Universal Robots PolyScope program: cb_pulley_v3.urp

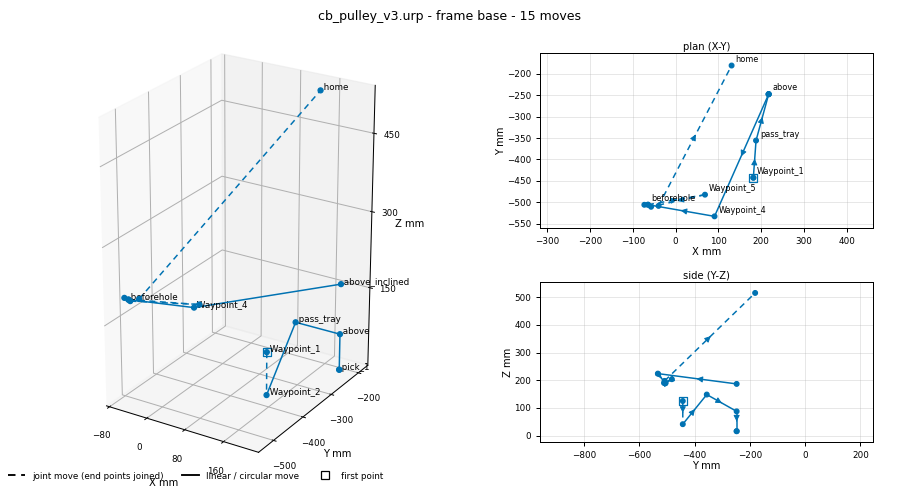
[picture p0: tool path of cb_pulley_v3.urp in frame base, 15 of 29 moves have a stored position in this frame; points joined in program order, loops and branches not executed]
Program cb_pulley_v3 (installation=default directory=/programs/wrs2020 createdIn=5.7.0.90932 lastSavedIn=5.10.0.106288 robotSerialNumber=20205500607)
Calibrated DH parameters: a=[0.000096, -0.337, -0.383372, 0.000118, 0.000015, 0]; d=[0.162724, 79.377998, -95.545185, 16.300583, 0.099689, 0.099499]; alpha=[1.569249, 0.003272, 0.005201, 1.570041, -1.570219, 0]; deltaTheta=[0, 0.65664, 5.410619, 0.215927, -0.000001, 0]
Robot Program (runOnlyOnce=true)
  Folder Center grasp
    MoveJ speed 60 deg/s, acceleration 80 deg/s^2 (useActiveTCP=true) feature=Base
      Waypoint Waypoint_1: TCP in base x=181.408 y=-442.546 z=124.895 mm, rx=-2.2287 ry=-2.203 rz=0.0809 rad; joints [97.762, -87.43, 118.13, -122.132, -92.283, 98.398] deg; TCP offset x=0 y=0 z=165 mm, rx=0 ry=0 rz=0 rad
      URCap Gripper (Robotiq_Grippers, Robotiq Inc.) dataModel(position=0.0, force=100.0, speed=100.0, positionInDouble=0.0, forceInDouble=100.0, speedInDouble=100.0, slaveIds=[9], blocking=true)
      Waypoint Waypoint_2: TCP in base x=181.416 y=-442.576 z=40.986 mm, rx=-2.2287 ry=-2.203 rz=0.081 rad; joints [97.73, -79.301, 124.264, -136.398, -92.298, 98.449] deg
      URCap Gripper (Robotiq_Grippers, Robotiq Inc.) dataModel(position=100.0, force=0.0, speed=0.0, positionInDouble=100.0, forceInDouble=0.0, speedInDouble=0.0, slaveIds=[9], blocking=true)
    MoveL speed 250 mm/s, acceleration 1200 mm/s^2 (useActiveTCP=true) feature=Base
      Waypoint pass_tray: TCP in base x=187.718 y=-355.766 z=148.266 mm, rx=0.1175 ry=3.1177 rz=-0.0239 rad; joints [97.948, -100.949, 126.425, -116.523, -88.651, 12.221] deg
      Waypoint above: motionParameters(blendRadius=0.05); TCP in base x=217.16 y=-247.644 z=87.424 mm, rx=1.2479 ry=2.8551 rz=-0.0099 rad; joints [106.845, -108.195, 141.669, -124.673, -88.866, 64.052] deg
      Waypoint pick_1: TCP in base x=217.16 y=-247.644 z=15.634 mm, rx=1.2479 ry=2.8551 rz=-0.0099 rad; joints [106.782, -96.811, 148.173, -142.561, -88.879, 64.086] deg
    URCap Gripper (Robotiq_Grippers, Robotiq Inc.) dataModel(position=27.45098039215686, force=100.0, speed=0.0, positionInDouble=27.45098039215686, forceInDouble=100.0, speedInDouble=0.0, slaveIds=[9], blocking=true)
    MoveL speed 800 mm/s, acceleration 1200 mm/s^2 (useActiveTCP=true) feature=Base
      Waypoint turn_left (Relative): relativeFromPosition TCP in base x=217.155 y=-247.662 z=15.637 mm, rx=1.248 ry=2.8551 rz=-0.0099 rad; joints [106.781, -96.81, 148.171, -142.561, -88.879, 64.086] deg; TCP in base x=217.136 y=-247.633 z=15.614 mm, rx=-1.1429 ry=2.9115 rz=-0.0354 rad; joints [106.78, -96.81, 148.175, -142.562, -88.881, -26] deg
    URCap Gripper (Robotiq_Grippers, Robotiq Inc.) dataModel(position=100.0, force=0.0, speed=0.0, positionInDouble=100.0, forceInDouble=0.0, speedInDouble=0.0, slaveIds=[9], blocking=true)
    URCap Gripper (Robotiq_Grippers, Robotiq Inc.) dataModel(position=36.07843137254902, force=100.0, speed=0.0, positionInDouble=36.07843137254902, forceInDouble=100.0, speedInDouble=0.0, slaveIds=[9], blocking=true)
    MoveL speed 800 mm/s, acceleration 1200 mm/s^2 (useActiveTCP=true) feature=Base
      Waypoint pick_1: TCP in base x=217.16 y=-247.644 z=15.634 mm, rx=1.2479 ry=2.8551 rz=-0.0099 rad; joints [106.782, -96.811, 148.173, -142.561, -88.879, 64.086] deg
      Waypoint incline (Relative): relativeFromPosition TCP in base x=128.749 y=-616.686 z=36.967 mm, rx=1.2364 ry=2.8602 rz=-0.0099 rad; joints [89.138, -62.117, 99.447, -128.197, -88.435, 45.998] deg; TCP in base x=123.207 y=-621.876 z=39.244 mm, rx=-1.1443 ry=-2.5469 rz=0.8367 rad; joints [100.881, -59.401, 111.689, -163.651, -118.976, 53.917] deg
    URCap Gripper (Robotiq_Grippers, Robotiq Inc.) dataModel(position=100.0, force=0.0, speed=100.0, positionInDouble=100.0, forceInDouble=0.0, speedInDouble=100.0, slaveIds=[9], blocking=true)
  MoveL speed 800 mm/s, acceleration 1200 mm/s^2 (useActiveTCP=true) feature=Base
    Waypoint above_inclined: motionParameters(blendRadius=0.05); TCP in base x=217.16 y=-247.644 z=186.776 mm, rx=1.2479 ry=2.8551 rz=-0.0099 rad; joints [106.918, -115.958, 130.039, -105.279, -88.87, 64.02] deg
    Waypoint Waypoint_4: motionParameters(blendRadius=0.05); TCP in base x=90.784 y=-532.798 z=224.095 mm, rx=1.3194 ry=-2.4664 rz=0.0869 rad; joints [93.539, -87.4, 107.422, -121.697, -105.954, -54.416] deg
    Waypoint beforehole: motionParameters(blendRadius=0); TCP in base x=-64.521 y=-505.594 z=189.248 mm, rx=1.6358 ry=-1.672 rz=-0.8845 rad; joints [92.147, -76.667, 111.26, -118.048, -144.223, -83.204] deg
  MoveL speed 20 mm/s, acceleration 1200 mm/s^2 (useActiveTCP=true) feature=Base
    Waypoint athole: TCP in base x=-73.031 y=-505.785 z=190.533 mm, rx=1.6339 ry=-1.6785 rz=-0.8787 rad; joints [91.13, -76.968, 111.703, -119.658, -144.069, -84.688] deg
  MoveL speed 20 mm/s, acceleration 1200 mm/s^2 (useActiveTCP=true) feature=Base
    MoveDirectionNode (selectedDirection=XMinus) feature=Base
      Until TOOL_CONTACT_DETECTION (allowActions=false retraction=0 decelerationAcceleration=3 decelerationAngularAcceleration=34.906585)
  Folder twist onto pin
    Force Frame feature=Base; selection=[1, 0, 0, 0, 0, 0]; wrench=[-10, 0, 0, 0, 0, 0]; limitsForce=[0.005, 0.01, 0.01, 1.047198, 1.047198, 1.047198]; limitsMotion=[0.1, 0.1, 0.1, 0.349066, 0.349066, 0.349066]
      MoveL speed 100 mm/s, acceleration 200 mm/s^2 (useActiveTCP=true) feature=Base
        Waypoint rightturn (Relative): relativeFromPosition TCP in base x=-72.572 y=-505.592 z=189.212 mm, rx=1.6359 ry=-1.672 rz=-0.8845 rad; joints [91.257, -76.786, 111.802, -119.705, -144.314, -84.72] deg; TCP in base x=-72.593 y=-509.312 z=189.314 mm, rx=1.2962 ry=-1.7188 rz=-0.4228 rad; joints [91.397, -77.772, 124.92, -159.613, -145.042, -84.31] deg
        Waypoint leftturn (Relative): relativeFromPosition TCP in base x=-72.61 y=-509.315 z=189.348 mm, rx=1.2962 ry=-1.7188 rz=-0.4228 rad; joints [91.396, -77.774, 124.918, -159.612, -145.044, -84.311] deg; TCP in base x=-72.577 y=-505.577 z=189.198 mm, rx=1.6359 ry=-1.6719 rz=-0.8846 rad; joints [91.257, -76.786, 111.804, -119.704, -144.316, -84.721] deg
        Waypoint leftturn (Relative): relativeFromPosition TCP in base x=-72.61 y=-509.315 z=189.348 mm, rx=1.2962 ry=-1.7188 rz=-0.4228 rad; joints [91.396, -77.774, 124.918, -159.612, -145.044, -84.311] deg; TCP in base x=-72.577 y=-505.577 z=189.198 mm, rx=1.6359 ry=-1.6719 rz=-0.8846 rad; joints [91.257, -76.786, 111.804, -119.704, -144.316, -84.721] deg
        Waypoint rightturn (Relative): relativeFromPosition TCP in base x=-72.572 y=-505.592 z=189.212 mm, rx=1.6359 ry=-1.672 rz=-0.8845 rad; joints [91.257, -76.786, 111.802, -119.705, -144.314, -84.72] deg; TCP in base x=-72.593 y=-509.312 z=189.314 mm, rx=1.2962 ry=-1.7188 rz=-0.4228 rad; joints [91.397, -77.772, 124.92, -159.613, -145.042, -84.31] deg
    tcp_p := get_actual_tcp_pose()
    SuppressedNode
      If tcp_p[0] > -0.08
        Force Frame feature=Base; selection=[1, 1, 1, 0, 0, 0]; wrench=[-10, 0, 0, 0, 0, 0]; limitsForce=[0.005, 0.002, 0.002, 1.047198, 1.047198, 1.047198]; limitsMotion=[0.1, 0.1, 0.1, 0.349066, 0.349066, 0.349066]
          MoveL speed 5 mm/s, acceleration 2 mm/s^2 (useActiveTCP=true) feature=Base
            MoveDirectionNode (selectedDirection=ZPlus) feature=Base
              Until DISTANCE (allowActions=false deceleration=3 distanceNodeType=STOP) Distance=0.001; motionParameters(blendRadius=0)
            MoveDirectionNode (selectedDirection=ZMinus) feature=Base
              Until DISTANCE (allowActions=false deceleration=3 distanceNodeType=STOP) Distance=0.002; motionParameters(blendRadius=0)
            MoveDirectionNode (selectedDirection=ZPlus) feature=Base
              Until DISTANCE (allowActions=false deceleration=3 distanceNodeType=STOP) Distance=0.001; motionParameters(blendRadius=0)
            MoveDirectionNode (selectedDirection=YPlus) feature=Base
              Until DISTANCE (allowActions=false deceleration=3 distanceNodeType=STOP) Distance=0.001; motionParameters(blendRadius=0)
            MoveDirectionNode (selectedDirection=YMinus) feature=Base
              Until DISTANCE (allowActions=false deceleration=3 distanceNodeType=STOP) Distance=0.002; motionParameters(blendRadius=0)
            MoveDirectionNode (selectedDirection=YPlus) feature=Base
              Until DISTANCE (allowActions=false deceleration=3 distanceNodeType=STOP) Distance=0.001; motionParameters(blendRadius=0)
    tcp_p := get_actual_tcp_pose()
    If tcp_p[0] > -0.08
      Force Frame feature=Base; selection=[1, 0, 0, 0, 0, 0]; wrench=[-40, 0, 0, 0, 0, 0]; limitsForce=[0.005, 0.01, 0.01, 1.047198, 1.047198, 1.047198]; limitsMotion=[0.1, 0.1, 0.1, 0.349066, 0.349066, 0.349066]
        MoveL speed 100 mm/s, acceleration 200 mm/s^2 (useActiveTCP=true) feature=Base
          Waypoint rightturn (Relative): relativeFromPosition TCP in base x=-72.572 y=-505.592 z=189.212 mm, rx=1.6359 ry=-1.672 rz=-0.8845 rad; joints [91.257, -76.786, 111.802, -119.705, -144.314, -84.72] deg; TCP in base x=-72.593 y=-509.312 z=189.314 mm, rx=1.2962 ry=-1.7188 rz=-0.4228 rad; joints [91.397, -77.772, 124.92, -159.613, -145.042, -84.31] deg
          Waypoint leftturn (Relative): relativeFromPosition TCP in base x=-72.61 y=-509.315 z=189.348 mm, rx=1.2962 ry=-1.7188 rz=-0.4228 rad; joints [91.396, -77.774, 124.918, -159.612, -145.044, -84.311] deg; TCP in base x=-72.577 y=-505.577 z=189.198 mm, rx=1.6359 ry=-1.6719 rz=-0.8846 rad; joints [91.257, -76.786, 111.804, -119.704, -144.316, -84.721] deg
          Waypoint leftturn (Relative): relativeFromPosition TCP in base x=-72.61 y=-509.315 z=189.348 mm, rx=1.2962 ry=-1.7188 rz=-0.4228 rad; joints [91.396, -77.774, 124.918, -159.612, -145.044, -84.311] deg; TCP in base x=-72.577 y=-505.577 z=189.198 mm, rx=1.6359 ry=-1.6719 rz=-0.8846 rad; joints [91.257, -76.786, 111.804, -119.704, -144.316, -84.721] deg
          Waypoint rightturn (Relative): relativeFromPosition TCP in base x=-72.572 y=-505.592 z=189.212 mm, rx=1.6359 ry=-1.672 rz=-0.8845 rad; joints [91.257, -76.786, 111.802, -119.705, -144.314, -84.72] deg; TCP in base x=-72.593 y=-509.312 z=189.314 mm, rx=1.2962 ry=-1.7188 rz=-0.4228 rad; joints [91.397, -77.772, 124.92, -159.613, -145.042, -84.31] deg
  URCap Gripper (Robotiq_Grippers, Robotiq Inc.) dataModel(position=0.0, force=100.0, speed=100.0, positionInDouble=0.0, forceInDouble=100.0, speedInDouble=100.0, slaveIds=[9], blocking=true)
  tcp_p := get_actual_tcp_pose()
  If tcp_p[0] > -0.09
    MoveJ speed 120 deg/s, acceleration 150 deg/s^2 (useActiveTCP=true) feature=Base
      Waypoint beforehole: TCP in base x=-64.521 y=-505.594 z=189.248 mm, rx=1.6358 ry=-1.672 rz=-0.8845 rad; joints [92.147, -76.667, 111.26, -118.048, -144.223, -83.204] deg
      URCap Gripper (Robotiq_Grippers, Robotiq Inc.) dataModel(position=74.11764705882352, force=100.0, speed=100.0, positionInDouble=74.11764705882352, forceInDouble=100.0, speedInDouble=100.0, slaveIds=[9], blocking=false)
      Waypoint Waypoint_5: motionParameters(blendRadius=0.05); TCP in base x=68.522 y=-482.203 z=203.802 mm, rx=1.8496 ry=-2.2565 rz=0.2806 rad; joints [82.53, -98.422, 121.376, -129.22, -89.967, -86.171] deg
      Waypoint Waypoint_8: TCP in base x=-57.337 y=-510.469 z=190.091 mm, rx=2.0055 ry=-2.1107 rz=0.242 rad; joints [66.732, -93.938, 119.294, -130.674, -85.997, -109.808] deg
    Folder push onto pin
      loop_1 := 1
      tcp_p := get_actual_tcp_pose()
      Force Frame feature=Base; selection=[1, 0, 0, 0, 0, 0]; wrench=[-40, 0, 0, 0, 0, 0]; limitsForce=[0.01, 0.01, 0.01, 1.047198, 1.047198, 1.047198]; limitsMotion=[0.1, 0.1, 0.1, 0.349066, 0.349066, 0.349066]
        Loop While (checkContinuously=true) expression=( tcp_p[0] > -0.090) and  (loop_1 < 3)
          MoveL speed 50 mm/s, acceleration 200 mm/s^2 (useActiveTCP=true) feature=Base
            Waypoint right1 (Relative): relativeFromPosition TCP in base x=-56.979 y=-508.359 z=197.636 mm, rx=1.9455 ry=-2.0777 rz=0.1274 rad; joints [70.294, -94.262, 119.256, -132.208, -92.762, -106.364] deg; TCP in base x=-56.977 y=-508.344 z=197.639 mm, rx=2.0958 ry=-1.919 rz=0.0946 rad; joints [70.293, -94.264, 119.256, -132.205, -92.762, -115.171] deg
            tcp_p := get_actual_tcp_pose()
            Waypoint left1 (Relative): relativeFromPosition TCP in base x=-56.985 y=-508.33 z=197.605 mm, rx=2.0958 ry=-1.919 rz=0.0945 rad; joints [70.293, -94.262, 119.258, -132.206, -92.764, -115.169] deg; TCP in base x=-56.968 y=-508.356 z=197.628 mm, rx=1.9456 ry=-2.0776 rz=0.1273 rad; joints [70.294, -94.261, 119.255, -132.205, -92.762, -106.365] deg
            tcp_p := get_actual_tcp_pose()
            Waypoint left1 (Relative): relativeFromPosition TCP in base x=-56.985 y=-508.33 z=197.605 mm, rx=2.0958 ry=-1.919 rz=0.0945 rad; joints [70.293, -94.262, 119.258, -132.206, -92.764, -115.169] deg; TCP in base x=-56.968 y=-508.356 z=197.628 mm, rx=1.9456 ry=-2.0776 rz=0.1273 rad; joints [70.294, -94.261, 119.255, -132.205, -92.762, -106.365] deg
            tcp_p := get_actual_tcp_pose()
            Waypoint right1 (Relative): relativeFromPosition TCP in base x=-56.979 y=-508.359 z=197.636 mm, rx=1.9455 ry=-2.0777 rz=0.1274 rad; joints [70.294, -94.262, 119.256, -132.208, -92.762, -106.364] deg; TCP in base x=-56.977 y=-508.344 z=197.639 mm, rx=2.0958 ry=-1.919 rz=0.0946 rad; joints [70.293, -94.264, 119.256, -132.205, -92.762, -115.171] deg
            tcp_p := get_actual_tcp_pose()
          loop_1 := loop_1+1
  MoveJ speed 60 deg/s, acceleration 80 deg/s^2 (useActiveTCP=true) feature=Base
    Waypoint back: TCP in base x=-39.842 y=-508.361 z=197.658 mm, rx=1.9455 ry=-2.0776 rz=0.1274 rad; joints [72.514, -94.336, 119.286, -132.039, -93.419, -104.24] deg
  MoveJ speed 180 deg/s, acceleration 80 deg/s^2 (useActiveTCP=true) feature=Base
    Waypoint home: TCP in base x=130.635 y=-180.692 z=515.97 mm, rx=-0.0117 ry=-3.1402 rz=-0.0315 rad; joints [89.951, -120.324, 80.212, -48.705, -89.957, -0.002] deg
